(*********************************** G.D S.p.A. - Technical Department ***********************************
============= PROGRAM INFO ============
FOLDER:             TBD
MACHINES INVOLVED:  TBD 

============= DESCRIPTION =============
csp machine declaration

============= REVISIONS ===============
Date		Version	 	Author      	Description             
----------	-------		------------  	--------------------------------------------
2019/04/05 	0000.00	 	M.Grasso		Creation of the PRG

**********************************************************************************************************)
(*$R process_ref := prc; $*)
PROGRAM csp_case_feed_arm_elbow
VAR
		
	prc:												process;
	prc_path:											STRING;
	
	axis:												axis;
	servo_on_condition:									BOOL;
	torque_limit:										INT := 2000;    (*$P $*)
	torque_limit_old:									INT;
	in_accu_safe_pos:                                   BOOL := FALSE;
    accu_tolerance:                                     INT := 5;
    accu_safe_pos:                                      INT;
    enable_delay:                                       TON;
	Torque_force_constant: 								LREAL := 1.31;
END_VAR

VAR CONSTANT
	MOTOR_MAX_VELOCITY_DEGPS:							LREAL := 9600;
	MOTOR_MAX_ACCELLERATION_DEGPS2:						LREAL := 4800;
	MOTOR_MAX_DECELLERATION_DEGPS2:						LREAL := 4800;
	MOTOR_MAX_JERK_DEGPS3:								LREAL := 100000000; 
	MOTOR_MAX_FOLLOWING_ERROR_DEG:						LREAL := 2;
END_VAR

_read_var_input();

_object_manager();

IF NOT objects_running()
THEN
	RETURN;	
END_IF

_read_process_image();

_mode_manager();

CASE process_get_mode(prc) OF
	MODE_ABSENT:
		IF axis_get_mode(axis) = MODE_TEST
		THEN
			safety_integrated_series_close(csp_case_main_safety_drives_SD8200.chA_smes_sis);
		END_IF
		RETURN;
	MODE_INACTIVE:
		RETURN;
	MODE_TEST:
		_handle_process_test();
END_CASE

_set_runtime_properties();

(********************************* BODY *********************************)
axis.actual_torque := (axis.actual_current * Torque_force_constant)/1000;

// Sets the torque limit for the case feed elbow
IF torque_limit <> Torque_limit_old
THEN
	 IF soe_drive_channel_write_parameter(
		channel:=csp_case_feed_arm_elbow.axis.soe_drive_channel, 
		idn:= S_0_IDN + 92, 
		data_element:=soe_drive_element_value , 
		data_source:= ADR(torque_limit), 
		data_lenght:= SIZEOF(torque_limit), 
		CONVERSION_this:= csp_case_feed_arm_elbow.axis.soe_drive^)= SOE_DRIVE_RETURN_VALUE_DONE
	THEN
		torque_limit_old := Torque_limit;
	END_IF
END_IF
(************************************************************************)

_handle_messages();

_write_output();

ACTION _handle_messages:
;
END_ACTION

ACTION _handle_process_test:
;
END_ACTION

ACTION _mode_manager:
IF process_mode_req_is_pending(prc)
THEN
    process_apply_mode_req_first_step(prc);
    CASE process_get_mode(prc) OF
        MODE_TO_ABSENT:
			;
        MODE_TO_INACTIVE:
			;
        MODE_TO_TEST:
			;
        MODE_TO_OPERATIONAL:
			;
    END_CASE
    process_apply_mode_req_second_step(prc);
END_IF
END_ACTION

ACTION _object_manager:
IF objects_initialization()
THEN
	sub_process_init(
		object_name									:= 'csp_case_feed_arm_elbow.prc', 
		process										:= csp_case_feed_arm.prc, 
		CONVERSION_this								:= prc);
		
	prc_path 										:= process_get_path(prc);
	
(* axis smes *)
	IF csp_main_configurator.Physical_hw
	THEN	
		axis_init(
			object_name								:= CONCAT(prc_path, '_axis'), 
			axis_type								:= AXIS_TYPE_SERVO, 
			encoder_scaling_factor					:= G_SERVO_ENCODER_SCALING_FACTOR_DEGPINC,
			modulo									:= G_NO_MODULO_DEG, 
			process									:= prc, 
			CONVERSION_this							:= axis);
			
		axis_add_safety_integrated_series(
			safety_integrated_series 				:= csp_case_main_safety_drives_SD8200.chA_smes_sis,
			CONVERSION_this							:= axis);
			
		axis_init_absolute_encoder_preset(
			position                                := 107,
			CONVERSION_this                         := axis);
			
			
	ELSE
		axis_init(
			object_name								:= CONCAT(prc_path, '_axis'), 
			axis_type								:= AXIS_TYPE_VIRTUAL, 
			encoder_scaling_factor					:= G_VIRTUAL_ENCODER_SCALING_FACTOR_DEGPINC,
			modulo									:= G_MODULO_360_DEG, 
			process									:= prc, 
			CONVERSION_this							:= axis);		
			
	END_IF
	
	axis_set_max_dynamic(
		reference_velocity							:=	MOTOR_MAX_VELOCITY_DEGPS,
		velocity									:=	MOTOR_MAX_VELOCITY_DEGPS,
		acceleration								:=	MOTOR_MAX_ACCELLERATION_DEGPS2,
		deceleration								:=	MOTOR_MAX_DECELLERATION_DEGPS2,
		jerk										:=	MOTOR_MAX_JERK_DEGPS3,
		following_error								:=	MOTOR_MAX_FOLLOWING_ERROR_DEG,
		CONVERSION_this								:=	axis);
		
	axis_add_soe_drive(
		channel										:=	SOE_DRIVE_CHANNEL_A,
		soe_drive									:=	csp_case_main_drives.SD8200_drv,
		CONVERSION_this								:=	axis);

			
END_IF

IF objects_running()
THEN
	process_cycle(prc);
	axis_cycle(axis);
END_IF
END_ACTION

ACTION _read_process_image:
;
END_ACTION

ACTION _read_var_input:
;
END_ACTION

ACTION _set_runtime_properties:
enable_delay(IN:=axis_is_ready_to_enable(axis) , PT:=T#2S , Q=> servo_on_condition , ET=> );
END_ACTION

ACTION _write_output:
;
END_ACTION

END_PROGRAM

(* stored: Version 1.1.0.1, ProductVersion 3.1.4024.3
   POU csp_case_feed_arm_elbow: Id {53eb0ad9-c05f-4ff4-9b79-820d9f94a238}, SpecialFunc None
   Action _handle_messages: Id {bb27c863-9746-40c3-a52c-d889eae2d949}
   Action _handle_process_test: Id {70b930a9-5063-458d-aefa-40ee5500b9ea}
   Action _mode_manager: Id {56321730-5b1c-46a1-bfa9-9e3835de2892}
   Action _object_manager: Id {b5c0ba38-a1fc-44b5-81f5-e9bd9e39ace5}
   Action _read_process_image: Id {4712fbf7-5595-4d55-b62b-2f0cf6d2cabf}
   Action _read_var_input: Id {b6da3fd1-da8c-4f84-804c-2889a32ac7af}
   Action _set_runtime_properties: Id {3ab303a9-16bd-450d-a405-7d19cfa79339}
   Action _write_output: Id {a2f23de9-141e-413b-bdc2-4a2728f9ffef} *)
